PROGRAM PRG_Compilation
VAR
END_VAR

END_PROGRAM

(* stored: Version 1.1.0.1, ProductVersion 3.1.4024.15
   POU PRG_Compilation: Id {c7b8d360-1f07-4d6a-b795-97ab52a4b56b}, SpecialFunc None *)
